TYPE typeHMIheader :
STRUCT
	
	stationstate: INT;
	stationstateColour:BOOL;
	homestate: INT; //home state for text list
	homestateColour: BOOL; //colour state of indicator

	anotherstate: BOOL;
	//faultstate: BOOL;
	//stationname: BOOL;
	flasher: BOOL;

	stationNameSelect: UINT; //station name selection
	cycleTypeFeedback: INT;
	
	isFaultState: BOOL; //colour change header
	FaultStateHeader: INT; //text change on header
	
	AnyStationFaultHeaderActive:BOOL;//colour change for global header
	AnyStationFaultHeader:INT; //text select for global header
	AnyStationFaultColour:DWORD; //background blue, alarm red or warning yellow
	isAnyFaultState: BOOL; //colour change header
	
	isWarningState: BOOL; //colour change header
	WarningStateHeader: INT; //text change on header
	
	AnyStationWarningHeaderActive:BOOL;//colour change for global header
	AnyStationWarningHeader:INT; //text select for global header
	AnyStationWarningColour:DWORD; //background blue, alarm red or warning yellow
	isAnyWarningState: BOOL; //colour change header







END_STRUCT
END_TYPE

(* stored: Version 1.1.0.1, ProductVersion 3.1.4024.11
   DUT typeHMIheader: Id {c95c4980-1ece-470b-964a-d85f7da56a0f} *)
